GLOBALCONSTANTS logiBUS_DI_Events (* logiBUS_DI constants *)
  (* Standard: 61499-1; Description: Copyright (c) 2024 HR Agrartechnik GmbH This program and the accompanying materials are made available under the terms of the Eclipse Public License 2.0 which is available at https://www.eclipse.org/legal/epl-2.0/ SPDX-License-Identifier: EPL-2.0 *)
  (* Version 1.0, 2024-01-25, Franz Höpfinger, HR Agrartechnik GmbH *)
  VAR_GLOBAL CONSTANT
    BUTTON_PRESS_DOWN : logiBUS_DI_Events_S := (EType := 0); (* Button pressed *)
    BUTTON_PRESS_UP : logiBUS_DI_Events_S := (EType := 1); (* Button released *)
    BUTTON_PRESS_REPEAT : logiBUS_DI_Events_S := (EType := 2); (* Button pressed repeat *)
    BUTTON_PRESS_REPEAT_DONE : logiBUS_DI_Events_S := (EType := 3); (* Button press repeat done *)
    BUTTON_SINGLE_CLICK : logiBUS_DI_Events_S := (EType := 4); (* Button single click *)
    BUTTON_DOUBLE_CLICK : logiBUS_DI_Events_S := (EType := 5); (* Button double click *)
    BUTTON_MULTIPLE_CLICK : logiBUS_DI_Events_S := (EType := 6); (* Button multiple click *)
    BUTTON_LONG_PRESS_START : logiBUS_DI_Events_S := (EType := 7); (* Button long press start *)
    BUTTON_LONG_PRESS_HOLD : logiBUS_DI_Events_S := (EType := 8); (* Button long press hold *)
    BUTTON_LONG_PRESS_UP : logiBUS_DI_Events_S := (EType := 9); (* Button long press up *)
    BUTTON_PRESS_END : logiBUS_DI_Events_S := (EType := 10); (* Button Press end *)
    BUTTON_EVENT_MAX : logiBUS_DI_Events_S := (EType := 11);
    BUTTON_NONE_PRESS : logiBUS_DI_Events_S := (EType := 12);
    Invalid : logiBUS_DI_Events_S := (EType := 255);
  END_VAR
END_GLOBALCONSTANTS
